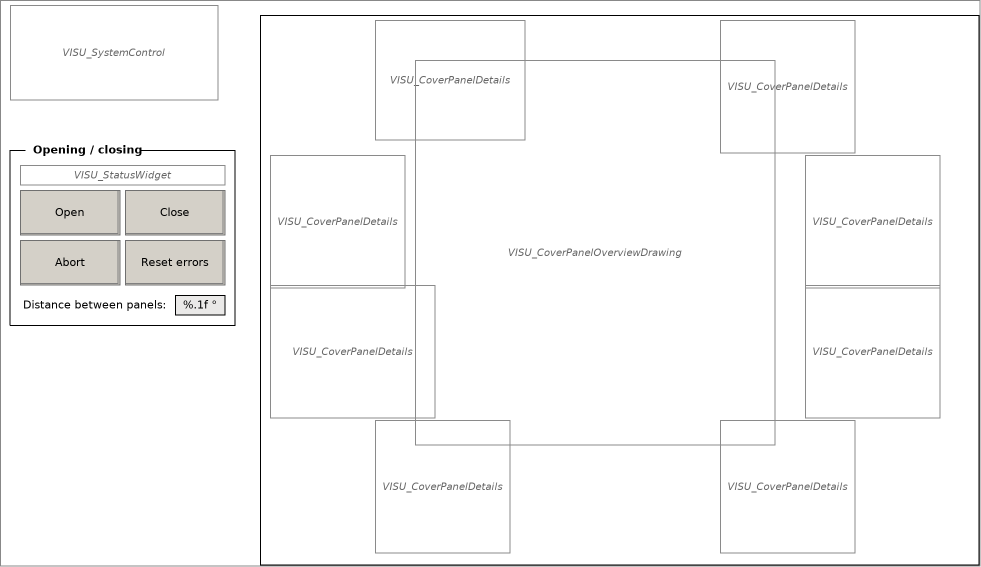
VISUALIZATION VISU_COVER_OVERVIEW  // 981x567
VAR_IN_OUT
	cover : Cover;
	coverWidget : CoverWidget;
END_VAR
    Rectangle (260,15 719x550)
    Frame (720,20 135x133)
        shows VISU_CoverPanelDetails(config := cover.config.top.p1, panel := cover.parts.top.parts.p1, widget := coverWidget.top.p1, magnetEnabled := cover.parts.top.parts.magnetsRelay.digitalOutput)
        pReferences[0]: name='Top 1'
    Frame (805,155 135x133)
        shows VISU_CoverPanelDetails(config := cover.config.bottom.p1, panel := cover.parts.bottom.parts.p1, widget := coverWidget.bottom.p1, magnetEnabled := cover.parts.bottom.parts.magnetsRelay.digitalOutput)
        pReferences[0]: name='Top 1'
    Frame (805,285 135x133)
        shows VISU_CoverPanelDetails(config := cover.config.top.p2, panel := cover.parts.top.parts.p2, widget := coverWidget.top.p2, magnetEnabled := cover.parts.top.parts.magnetsRelay.digitalOutput)
        pReferences[0]: name='Top 1'
    Frame (720,420 135x133)
        shows VISU_CoverPanelDetails(config := cover.config.bottom.p2, panel := cover.parts.bottom.parts.p2, widget := coverWidget.bottom.p2, magnetEnabled := cover.parts.bottom.parts.magnetsRelay.digitalOutput)
        pReferences[0]: name='Top 1'
    Frame (375,20 150x120)
        shows VISU_CoverPanelDetails(config := cover.config.bottom.p4, panel := cover.parts.bottom.parts.p4, widget := coverWidget.bottom.p4, magnetEnabled := cover.parts.bottom.parts.magnetsRelay.digitalOutput)
        pReferences[0]: name='Top 1'
    Frame (270,155 135x133)
        shows VISU_CoverPanelDetails(config := cover.config.top.p4, panel := cover.parts.top.parts.p4, widget := coverWidget.top.p4, magnetEnabled := cover.parts.top.parts.magnetsRelay.digitalOutput)
        pReferences[0]: name='Top 1'
    Frame (270,285 165x133)
        shows VISU_CoverPanelDetails(config := cover.config.bottom.p3, panel := cover.parts.bottom.parts.p3, widget := coverWidget.bottom.p3, magnetEnabled := cover.parts.bottom.parts.magnetsRelay.digitalOutput)
        pReferences[0]: name='Top 1'
    Frame (375,420 135x133)
        shows VISU_CoverPanelDetails(config := cover.config.top.p3, panel := cover.parts.top.parts.p3, widget := coverWidget.top.p3, magnetEnabled := cover.parts.top.parts.magnetsRelay.digitalOutput)
        pReferences[0]: name='Top 1'
    Frame (415,60 360x385)
        shows VISU_CoverPanelOverviewDrawing(cover := cover, coverWidget := coverWidget)
    Frame (10,5 208x95)
        shows VISU_SystemControl(status := coverWidget.actualStatus, button_initialize := coverWidget.button_initialize, button_operating := coverWidget.button_operating, button_locking := coverWidget.button_locking)
    Frame (20,165 205x20)
        shows VISU_StatusWidget(widget := coverWidget.apertureProcedureStatus)
    Button (20,190 100x45), "Open", input disabled if: cover.processes.open.statuses.enabledStatus.disabled
        OnMouseClick: execute { cover.processes.open.do_request := TRUE; }
    Button (125,190 100x45), "Close", input disabled if: cover.processes.close.statuses.enabledStatus.disabled
        OnMouseClick: execute { cover.processes.close.do_request := TRUE; }
    Button (20,240 100x45), "Abort", input disabled if: cover.processes.abort.statuses.enabledStatus.disabled
        OnMouseClick: execute { cover.processes.abort.do_request := TRUE; }
    Button (125,240 100x45), "Reset errors", input disabled if: cover.processes.reset.statuses.enabledStatus.disabled
        OnMouseClick: execute { cover.processes.reset.do_request := TRUE; }
    Rectangle (175,295 50x20), "%.1f °", text variable: cover.parts.apertureProcedure.distance.degrees.value
    Label (20,290 150x30), "Distance between panels:"
    Line (10,150) (25,150)
    Label (30,140 105x20), "Opening / closing"
    Line (140,150) (235,150)
    Line (235,325) (235,150)
    Line (10,325) (10,150)
    Line (10,325) (235,325)
END_VISUALIZATION

(* stored: Version 1.1.0.1, ProductVersion 3.1.4019.2
   Visu VISU_COVER_OVERVIEW: Id {00d2aea1-94f1-438a-8975-bd43a29a9dbf} *)
